TYPE T_Char : STRING[1];
END_TYPE

(* stored: Version 1.1.0.1, ProductVersion 3.1.4024.15
   DUT T_Char: Id {68c91db3-8b82-4a40-abbe-825d1b04bb7e} *)
